// TIA Portal V20 export
FUNCTION "02 T1-A ARUNC HMI" : Void   // FC1202, LAD
TITLE = HMI
{ S7_Optimized_Access := 'TRUE' }
// stored: AutoNumber false, SetENOAutomatically false
BEGIN

REGION Network 1: Reset command interface from HMI in case of time-out
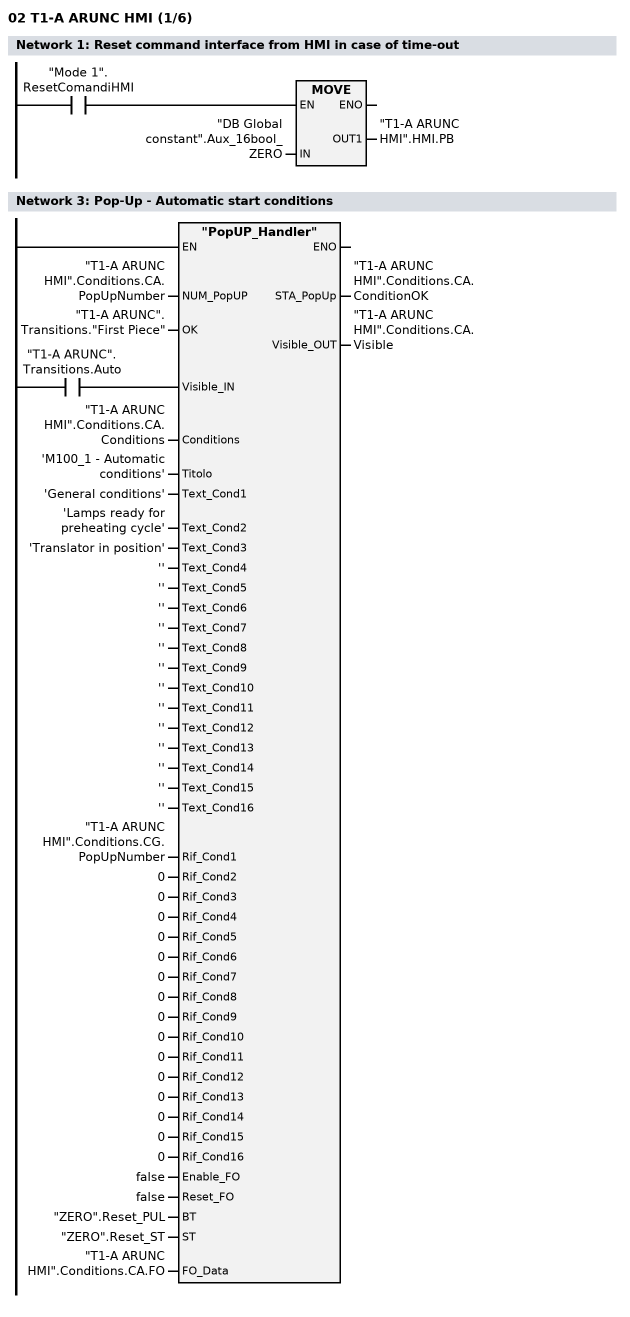
   RUNG wire#powerrail
      Contact( "Mode 1".ResetComandiHMI )
      Move(in := "DB Global constant".Aux_16bool_ZERO, out1 => "T1-A ARUNC HMI".HMI.PB)
   END_RUNG
   // the same network as SCL:
   IF "Mode 1".ResetComandiHMI THEN "T1-A ARUNC HMI".HMI.PB := "DB Global constant".Aux_16bool_ZERO; END_IF;
END_REGION

REGION Network 2: ============ POP UP ============
END_REGION

REGION Network 3: Pop-Up - Automatic start conditions
   RUNG wire#powerrail
      "PopUP_Handler"(Visible_IN := wire#w1, NUM_PopUP := "T1-A ARUNC HMI".Conditions.CA.PopUpNumber, OK := "T1-A ARUNC".Transitions."First Piece", Conditions := "T1-A ARUNC HMI".Conditions.CA.Conditions, Titolo := 'M100_1 - Automatic conditions', Text_Cond1 := 'General conditions', Text_Cond2 := 'Lamps ready for preheating cycle', Text_Cond3 := 'Translator in position', Text_Cond4 := '', Text_Cond5 := '', Text_Cond6 := '', Text_Cond7 := '', Text_Cond8 := '', Text_Cond9 := '', Text_Cond10 := '', Text_Cond11 := '', Text_Cond12 := '', Text_Cond13 := '', Text_Cond14 := '', Text_Cond15 := '', Text_Cond16 := '', Rif_Cond1 := "T1-A ARUNC HMI".Conditions.CG.PopUpNumber, Rif_Cond2 := 0, Rif_Cond3 := 0, Rif_Cond4 := 0, Rif_Cond5 := 0, Rif_Cond6 := 0, Rif_Cond7 := 0, Rif_Cond8 := 0, Rif_Cond9 := 0, Rif_Cond10 := 0, Rif_Cond11 := 0, Rif_Cond12 := 0, Rif_Cond13 := 0, Rif_Cond14 := 0, Rif_Cond15 := 0, Rif_Cond16 := 0, Enable_FO := false, Reset_FO := false, BT := "ZERO".Reset_PUL, ST := "ZERO".Reset_ST, FO_Data := "T1-A ARUNC HMI".Conditions.CA.FO, STA_PopUp => "T1-A ARUNC HMI".Conditions.CA.ConditionOK, Visible_OUT => "T1-A ARUNC HMI".Conditions.CA.Visible)
   END_RUNG
   RUNG wire#powerrail
      Contact( "T1-A ARUNC".Transitions.Auto )
   END_RUNG wire#w1
   // the same network as SCL:
   "PopUP_Handler"(NUM_PopUP := "T1-A ARUNC HMI".Conditions.CA.PopUpNumber,
                   OK := "T1-A ARUNC".Transitions."First Piece",
                   Visible_IN := "T1-A ARUNC".Transitions.Auto,
                   Conditions := "T1-A ARUNC HMI".Conditions.CA.Conditions,
                   Titolo := 'M100_1 - Automatic conditions',
                   Text_Cond1 := 'General conditions',
                   Text_Cond2 := 'Lamps ready for preheating cycle',
                   Text_Cond3 := 'Translator in position',
                   Text_Cond4 := '',
                   Text_Cond5 := '',
                   Text_Cond6 := '',
                   Text_Cond7 := '',
                   Text_Cond8 := '',
                   Text_Cond9 := '',
                   Text_Cond10 := '',
                   Text_Cond11 := '',
                   Text_Cond12 := '',
                   Text_Cond13 := '',
                   Text_Cond14 := '',
                   Text_Cond15 := '',
                   Text_Cond16 := '',
                   Rif_Cond1 := "T1-A ARUNC HMI".Conditions.CG.PopUpNumber,
                   Rif_Cond2 := 0,
                   Rif_Cond3 := 0,
                   Rif_Cond4 := 0,
                   Rif_Cond5 := 0,
                   Rif_Cond6 := 0,
                   Rif_Cond7 := 0,
                   Rif_Cond8 := 0,
                   Rif_Cond9 := 0,
                   Rif_Cond10 := 0,
                   Rif_Cond11 := 0,
                   Rif_Cond12 := 0,
                   Rif_Cond13 := 0,
                   Rif_Cond14 := 0,
                   Rif_Cond15 := 0,
                   Rif_Cond16 := 0,
                   Enable_FO := false,
                   Reset_FO := false,
                   BT := "ZERO".Reset_PUL,
                   ST := "ZERO".Reset_ST,
                   FO_Data := "T1-A ARUNC HMI".Conditions.CA.FO,
                   STA_PopUp => "T1-A ARUNC HMI".Conditions.CA.ConditionOK,
                   Visible_OUT => "T1-A ARUNC HMI".Conditions.CA.Visible);
END_REGION

REGION Network 4: Pop- Up - General conditions
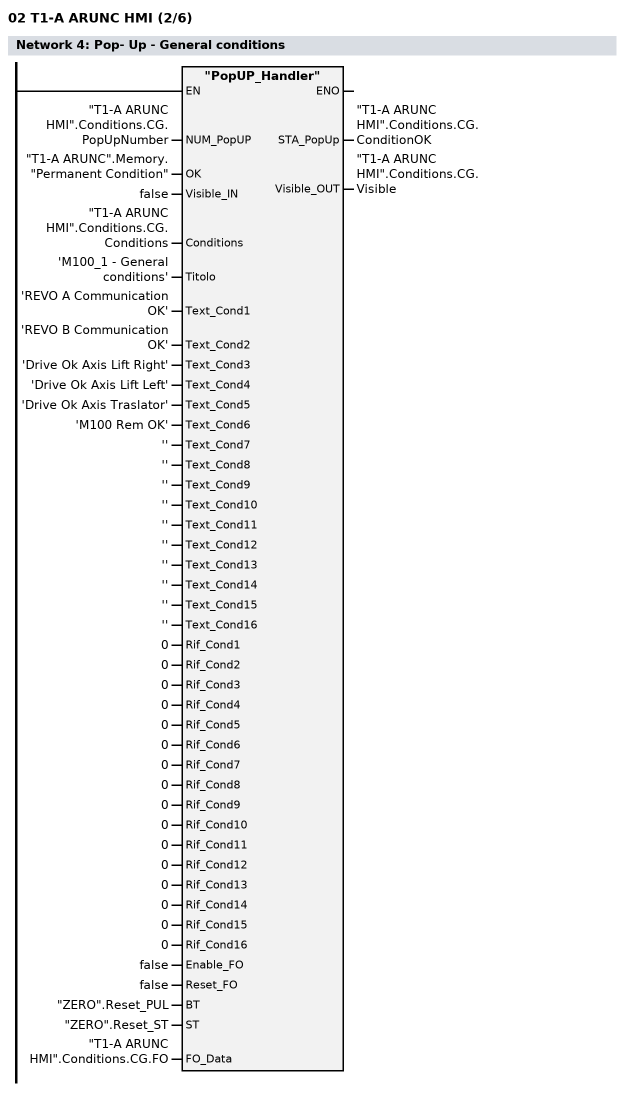
   RUNG wire#powerrail
      "PopUP_Handler"(NUM_PopUP := "T1-A ARUNC HMI".Conditions.CG.PopUpNumber, OK := "T1-A ARUNC".Memory."Permanent Condition", Visible_IN := false, Conditions := "T1-A ARUNC HMI".Conditions.CG.Conditions, Titolo := 'M100_1 - General conditions', Text_Cond1 := 'REVO A Communication OK', Text_Cond2 := 'REVO B Communication OK', Text_Cond3 := 'Drive Ok Axis Lift Right', Text_Cond4 := 'Drive Ok Axis Lift Left', Text_Cond5 := 'Drive Ok Axis Traslator', Text_Cond6 := 'M100 Rem OK', Text_Cond7 := '', Text_Cond8 := '', Text_Cond9 := '', Text_Cond10 := '', Text_Cond11 := '', Text_Cond12 := '', Text_Cond13 := '', Text_Cond14 := '', Text_Cond15 := '', Text_Cond16 := '', Rif_Cond1 := 0, Rif_Cond2 := 0, Rif_Cond3 := 0, Rif_Cond4 := 0, Rif_Cond5 := 0, Rif_Cond6 := 0, Rif_Cond7 := 0, Rif_Cond8 := 0, Rif_Cond9 := 0, Rif_Cond10 := 0, Rif_Cond11 := 0, Rif_Cond12 := 0, Rif_Cond13 := 0, Rif_Cond14 := 0, Rif_Cond15 := 0, Rif_Cond16 := 0, Enable_FO := false, Reset_FO := false, BT := "ZERO".Reset_PUL, ST := "ZERO".Reset_ST, FO_Data := "T1-A ARUNC HMI".Conditions.CG.FO, STA_PopUp => "T1-A ARUNC HMI".Conditions.CG.ConditionOK, Visible_OUT => "T1-A ARUNC HMI".Conditions.CG.Visible)
   END_RUNG
   // the same network as SCL:
   "PopUP_Handler"(NUM_PopUP := "T1-A ARUNC HMI".Conditions.CG.PopUpNumber,
                   OK := "T1-A ARUNC".Memory."Permanent Condition",
                   Visible_IN := false,
                   Conditions := "T1-A ARUNC HMI".Conditions.CG.Conditions,
                   Titolo := 'M100_1 - General conditions',
                   Text_Cond1 := 'REVO A Communication OK',
                   Text_Cond2 := 'REVO B Communication OK',
                   Text_Cond3 := 'Drive Ok Axis Lift Right',
                   Text_Cond4 := 'Drive Ok Axis Lift Left',
                   Text_Cond5 := 'Drive Ok Axis Traslator',
                   Text_Cond6 := 'M100 Rem OK',
                   Text_Cond7 := '',
                   Text_Cond8 := '',
                   Text_Cond9 := '',
                   Text_Cond10 := '',
                   Text_Cond11 := '',
                   Text_Cond12 := '',
                   Text_Cond13 := '',
                   Text_Cond14 := '',
                   Text_Cond15 := '',
                   Text_Cond16 := '',
                   Rif_Cond1 := 0,
                   Rif_Cond2 := 0,
                   Rif_Cond3 := 0,
                   Rif_Cond4 := 0,
                   Rif_Cond5 := 0,
                   Rif_Cond6 := 0,
                   Rif_Cond7 := 0,
                   Rif_Cond8 := 0,
                   Rif_Cond9 := 0,
                   Rif_Cond10 := 0,
                   Rif_Cond11 := 0,
                   Rif_Cond12 := 0,
                   Rif_Cond13 := 0,
                   Rif_Cond14 := 0,
                   Rif_Cond15 := 0,
                   Rif_Cond16 := 0,
                   Enable_FO := false,
                   Reset_FO := false,
                   BT := "ZERO".Reset_PUL,
                   ST := "ZERO".Reset_ST,
                   FO_Data := "T1-A ARUNC HMI".Conditions.CG.FO,
                   STA_PopUp => "T1-A ARUNC HMI".Conditions.CG.ConditionOK,
                   Visible_OUT => "T1-A ARUNC HMI".Conditions.CG.Visible);
END_REGION

REGION Network 5: PopUP - Cycle start conditions
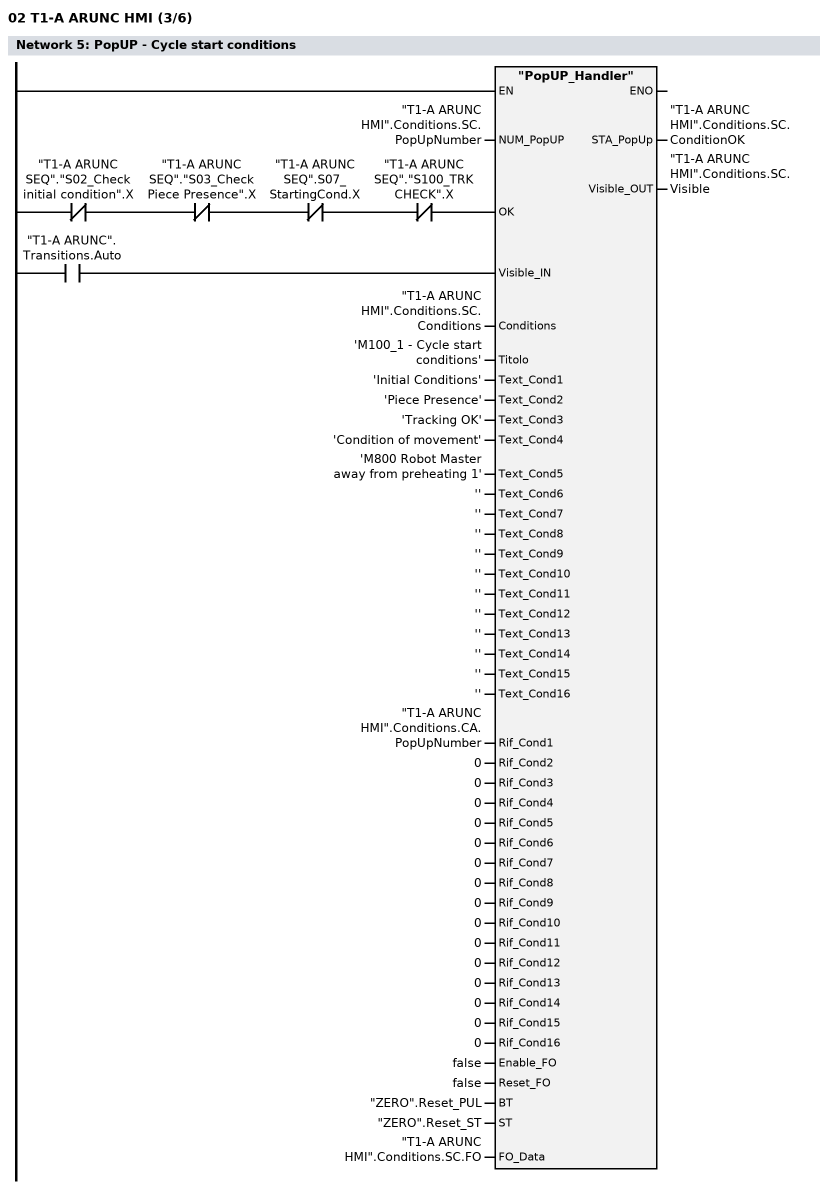
   RUNG wire#powerrail
      "PopUP_Handler"(OK := wire#w1, Visible_IN := wire#w2, NUM_PopUP := "T1-A ARUNC HMI".Conditions.SC.PopUpNumber, Conditions := "T1-A ARUNC HMI".Conditions.SC.Conditions, Titolo := 'M100_1 - Cycle start conditions', Text_Cond1 := 'Initial Conditions', Text_Cond2 := 'Piece Presence', Text_Cond3 := 'Tracking OK', Text_Cond4 := 'Condition of movement', Text_Cond5 := 'M800 Robot Master away from preheating 1', Text_Cond6 := '', Text_Cond7 := '', Text_Cond8 := '', Text_Cond9 := '', Text_Cond10 := '', Text_Cond11 := '', Text_Cond12 := '', Text_Cond13 := '', Text_Cond14 := '', Text_Cond15 := '', Text_Cond16 := '', Rif_Cond1 := "T1-A ARUNC HMI".Conditions.CA.PopUpNumber, Rif_Cond2 := 0, Rif_Cond3 := 0, Rif_Cond4 := 0, Rif_Cond5 := 0, Rif_Cond6 := 0, Rif_Cond7 := 0, Rif_Cond8 := 0, Rif_Cond9 := 0, Rif_Cond10 := 0, Rif_Cond11 := 0, Rif_Cond12 := 0, Rif_Cond13 := 0, Rif_Cond14 := 0, Rif_Cond15 := 0, Rif_Cond16 := 0, Enable_FO := false, Reset_FO := false, BT := "ZERO".Reset_PUL, ST := "ZERO".Reset_ST, FO_Data := "T1-A ARUNC HMI".Conditions.SC.FO, STA_PopUp => "T1-A ARUNC HMI".Conditions.SC.ConditionOK, Visible_OUT => "T1-A ARUNC HMI".Conditions.SC.Visible)
   END_RUNG
   RUNG wire#powerrail
      I_Contact( "T1-A ARUNC SEQ"."S02_Check initial condition".X )
      I_Contact( "T1-A ARUNC SEQ"."S03_Check Piece Presence".X )
      I_Contact( "T1-A ARUNC SEQ".S07_StartingCond.X )
      I_Contact( "T1-A ARUNC SEQ"."S100_TRK CHECK".X )
   END_RUNG wire#w1
   RUNG wire#powerrail
      Contact( "T1-A ARUNC".Transitions.Auto )
   END_RUNG wire#w2
   // the same network as SCL:
   "PopUP_Handler"(NUM_PopUP := "T1-A ARUNC HMI".Conditions.SC.PopUpNumber,
                   OK := NOT "T1-A ARUNC SEQ"."S02_Check initial condition".X AND NOT "T1-A ARUNC SEQ"."S03_Check Piece Presence".X AND NOT "T1-A ARUNC SEQ".S07_StartingCond.X AND NOT "T1-A ARUNC SEQ"."S100_TRK CHECK".X,
                   Visible_IN := "T1-A ARUNC".Transitions.Auto,
                   Conditions := "T1-A ARUNC HMI".Conditions.SC.Conditions,
                   Titolo := 'M100_1 - Cycle start conditions',
                   Text_Cond1 := 'Initial Conditions',
                   Text_Cond2 := 'Piece Presence',
                   Text_Cond3 := 'Tracking OK',
                   Text_Cond4 := 'Condition of movement',
                   Text_Cond5 := 'M800 Robot Master away from preheating 1',
                   Text_Cond6 := '',
                   Text_Cond7 := '',
                   Text_Cond8 := '',
                   Text_Cond9 := '',
                   Text_Cond10 := '',
                   Text_Cond11 := '',
                   Text_Cond12 := '',
                   Text_Cond13 := '',
                   Text_Cond14 := '',
                   Text_Cond15 := '',
                   Text_Cond16 := '',
                   Rif_Cond1 := "T1-A ARUNC HMI".Conditions.CA.PopUpNumber,
                   Rif_Cond2 := 0,
                   Rif_Cond3 := 0,
                   Rif_Cond4 := 0,
                   Rif_Cond5 := 0,
                   Rif_Cond6 := 0,
                   Rif_Cond7 := 0,
                   Rif_Cond8 := 0,
                   Rif_Cond9 := 0,
                   Rif_Cond10 := 0,
                   Rif_Cond11 := 0,
                   Rif_Cond12 := 0,
                   Rif_Cond13 := 0,
                   Rif_Cond14 := 0,
                   Rif_Cond15 := 0,
                   Rif_Cond16 := 0,
                   Enable_FO := false,
                   Reset_FO := false,
                   BT := "ZERO".Reset_PUL,
                   ST := "ZERO".Reset_ST,
                   FO_Data := "T1-A ARUNC HMI".Conditions.SC.FO,
                   STA_PopUp => "T1-A ARUNC HMI".Conditions.SC.ConditionOK,
                   Visible_OUT => "T1-A ARUNC HMI".Conditions.SC.Visible);
END_REGION

REGION Network 6: Pop-Up - Conditions of movement UP
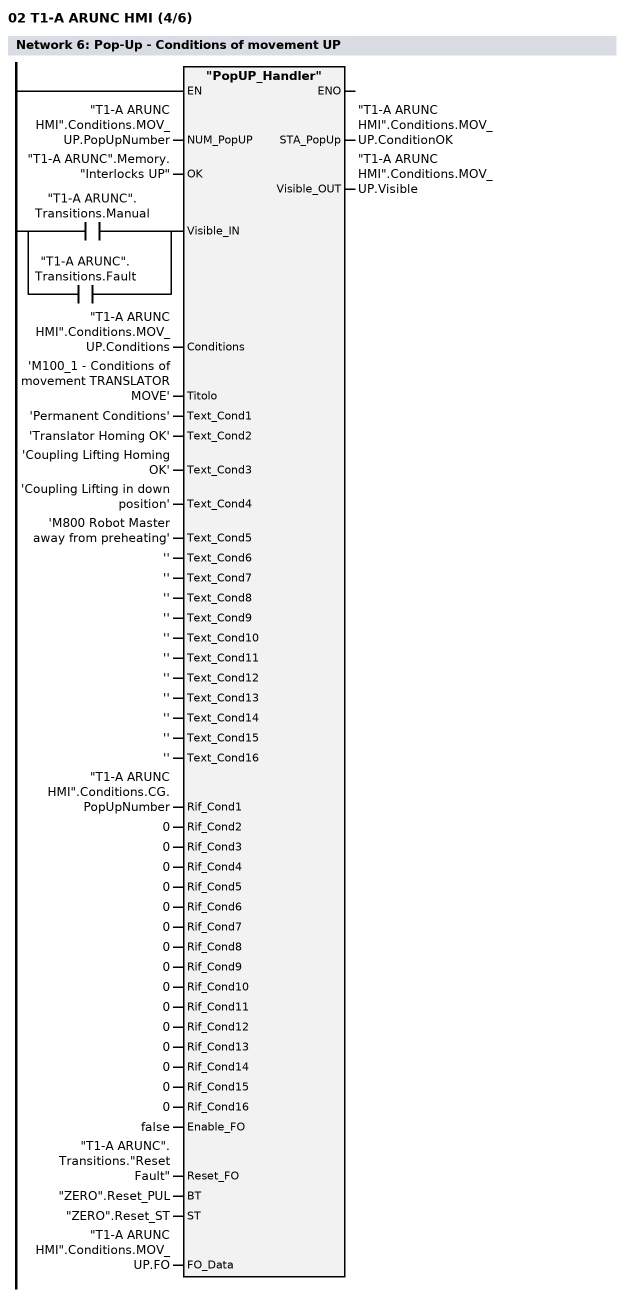
   RUNG wire#powerrail
      "PopUP_Handler"(Visible_IN := wire#w1, NUM_PopUP := "T1-A ARUNC HMI".Conditions.MOV_UP.PopUpNumber, OK := "T1-A ARUNC".Memory."Interlocks UP", Conditions := "T1-A ARUNC HMI".Conditions.MOV_UP.Conditions, Titolo := 'M100_1 - Conditions of movement TRANSLATOR MOVE', Text_Cond1 := 'Permanent Conditions', Text_Cond2 := 'Translator Homing OK', Text_Cond3 := 'Coupling Lifting Homing OK', Text_Cond4 := 'Coupling Lifting in down position', Text_Cond5 := 'M800 Robot Master away from preheating', Text_Cond6 := '', Text_Cond7 := '', Text_Cond8 := '', Text_Cond9 := '', Text_Cond10 := '', Text_Cond11 := '', Text_Cond12 := '', Text_Cond13 := '', Text_Cond14 := '', Text_Cond15 := '', Text_Cond16 := '', Rif_Cond1 := "T1-A ARUNC HMI".Conditions.CG.PopUpNumber, Rif_Cond2 := 0, Rif_Cond3 := 0, Rif_Cond4 := 0, Rif_Cond5 := 0, Rif_Cond6 := 0, Rif_Cond7 := 0, Rif_Cond8 := 0, Rif_Cond9 := 0, Rif_Cond10 := 0, Rif_Cond11 := 0, Rif_Cond12 := 0, Rif_Cond13 := 0, Rif_Cond14 := 0, Rif_Cond15 := 0, Rif_Cond16 := 0, Enable_FO := false, Reset_FO := "T1-A ARUNC".Transitions."Reset Fault", BT := "ZERO".Reset_PUL, ST := "ZERO".Reset_ST, FO_Data := "T1-A ARUNC HMI".Conditions.MOV_UP.FO, STA_PopUp => "T1-A ARUNC HMI".Conditions.MOV_UP.ConditionOK, Visible_OUT => "T1-A ARUNC HMI".Conditions.MOV_UP.Visible)
   END_RUNG
   RUNG wire#powerrail
      Contact( "T1-A ARUNC".Transitions.Manual )
   END_RUNG wire#w1
   RUNG wire#powerrail
      Contact( "T1-A ARUNC".Transitions.Fault )
   END_RUNG wire#w1
   // the same network as SCL:
   "PopUP_Handler"(NUM_PopUP := "T1-A ARUNC HMI".Conditions.MOV_UP.PopUpNumber,
                   OK := "T1-A ARUNC".Memory."Interlocks UP",
                   Visible_IN := "T1-A ARUNC".Transitions.Manual OR "T1-A ARUNC".Transitions.Fault,
                   Conditions := "T1-A ARUNC HMI".Conditions.MOV_UP.Conditions,
                   Titolo := 'M100_1 - Conditions of movement TRANSLATOR MOVE',
                   Text_Cond1 := 'Permanent Conditions',
                   Text_Cond2 := 'Translator Homing OK',
                   Text_Cond3 := 'Coupling Lifting Homing OK',
                   Text_Cond4 := 'Coupling Lifting in down position',
                   Text_Cond5 := 'M800 Robot Master away from preheating',
                   Text_Cond6 := '',
                   Text_Cond7 := '',
                   Text_Cond8 := '',
                   Text_Cond9 := '',
                   Text_Cond10 := '',
                   Text_Cond11 := '',
                   Text_Cond12 := '',
                   Text_Cond13 := '',
                   Text_Cond14 := '',
                   Text_Cond15 := '',
                   Text_Cond16 := '',
                   Rif_Cond1 := "T1-A ARUNC HMI".Conditions.CG.PopUpNumber,
                   Rif_Cond2 := 0,
                   Rif_Cond3 := 0,
                   Rif_Cond4 := 0,
                   Rif_Cond5 := 0,
                   Rif_Cond6 := 0,
                   Rif_Cond7 := 0,
                   Rif_Cond8 := 0,
                   Rif_Cond9 := 0,
                   Rif_Cond10 := 0,
                   Rif_Cond11 := 0,
                   Rif_Cond12 := 0,
                   Rif_Cond13 := 0,
                   Rif_Cond14 := 0,
                   Rif_Cond15 := 0,
                   Rif_Cond16 := 0,
                   Enable_FO := false,
                   Reset_FO := "T1-A ARUNC".Transitions."Reset Fault",
                   BT := "ZERO".Reset_PUL,
                   ST := "ZERO".Reset_ST,
                   FO_Data := "T1-A ARUNC HMI".Conditions.MOV_UP.FO,
                   STA_PopUp => "T1-A ARUNC HMI".Conditions.MOV_UP.ConditionOK,
                   Visible_OUT => "T1-A ARUNC HMI".Conditions.MOV_UP.Visible);
END_REGION

REGION Network 7: ============ HMI STATE ============
END_REGION

REGION Network 8: HMI Status - Aruncator
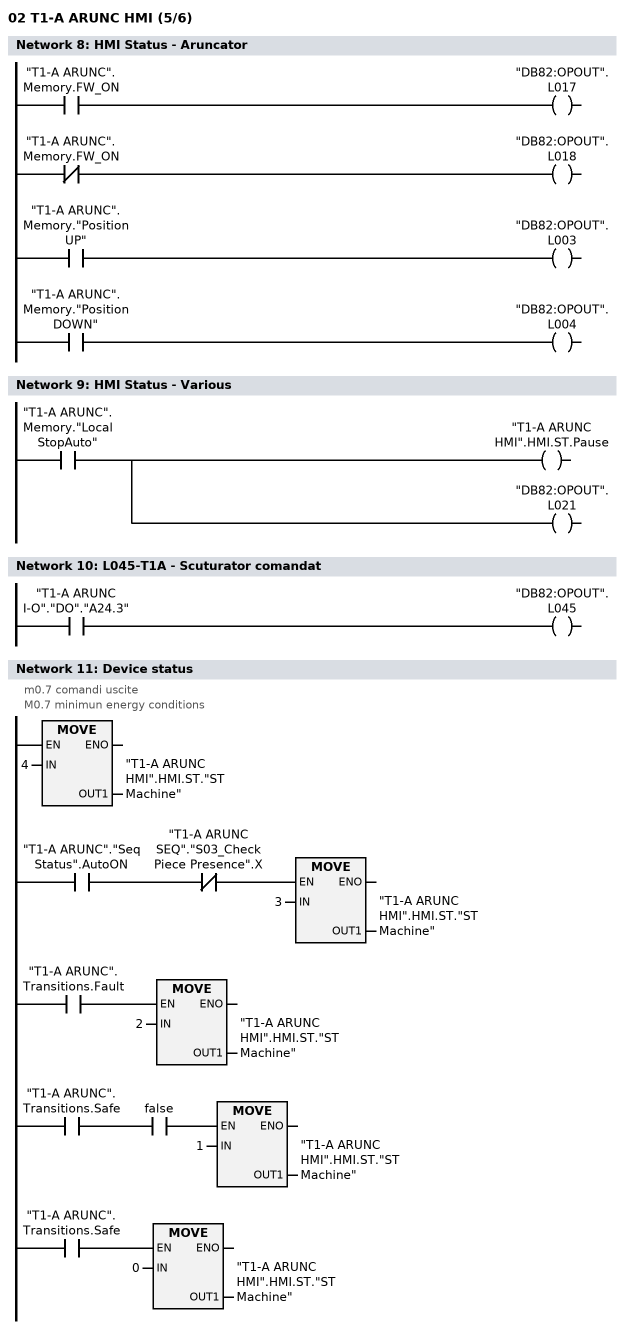
   RUNG wire#powerrail
      Contact( "T1-A ARUNC".Memory.FW_ON )
      Coil( "DB82:OPOUT".L017 )
   END_RUNG
   RUNG wire#powerrail
      I_Contact( "T1-A ARUNC".Memory.FW_ON )
      Coil( "DB82:OPOUT".L018 )
   END_RUNG
   RUNG wire#powerrail
      Contact( "T1-A ARUNC".Memory."Position UP" )
      Coil( "DB82:OPOUT".L003 )
   END_RUNG
   RUNG wire#powerrail
      Contact( "T1-A ARUNC".Memory."Position DOWN" )
      Coil( "DB82:OPOUT".L004 )
   END_RUNG
   // the same network as SCL:
   "DB82:OPOUT".L017 := "T1-A ARUNC".Memory.FW_ON;
   "DB82:OPOUT".L018 := NOT "T1-A ARUNC".Memory.FW_ON;
   "DB82:OPOUT".L003 := "T1-A ARUNC".Memory."Position UP";
   "DB82:OPOUT".L004 := "T1-A ARUNC".Memory."Position DOWN";
END_REGION

REGION Network 9: HMI Status - Various
   RUNG wire#powerrail
      Contact( "T1-A ARUNC".Memory."Local StopAuto" )
      wire#w1
      Coil( "T1-A ARUNC HMI".HMI.ST.Pause )
   END_RUNG
   RUNG wire#w1
      Coil( "DB82:OPOUT".L021 )
   END_RUNG
   // the same network as SCL:
   "T1-A ARUNC HMI".HMI.ST.Pause := "T1-A ARUNC".Memory."Local StopAuto";
   "DB82:OPOUT".L021 := "T1-A ARUNC".Memory."Local StopAuto";
END_REGION

REGION Network 10: L045-T1A - Scuturator comandat
   RUNG wire#powerrail
      Contact( "T1-A ARUNC I-O"."DO"."A24.3" )
      Coil( "DB82:OPOUT".L045 )
   END_RUNG
   // the same network as SCL:
   "DB82:OPOUT".L045 := "T1-A ARUNC I-O"."DO"."A24.3";
END_REGION

REGION Network 11: Device status
   // m0.7 comandi uscite
   // M0.7 minimun energy conditions
   RUNG wire#powerrail
      Move(in := 4, out1 => "T1-A ARUNC HMI".HMI.ST."ST Machine")
   END_RUNG
   RUNG wire#powerrail
      Contact( "T1-A ARUNC"."Seq Status".AutoON )
      I_Contact( "T1-A ARUNC SEQ"."S03_Check Piece Presence".X )
      Move(in := 3, out1 => "T1-A ARUNC HMI".HMI.ST."ST Machine")
   END_RUNG
   RUNG wire#powerrail
      Contact( "T1-A ARUNC".Transitions.Fault )
      Move(in := 2, out1 => "T1-A ARUNC HMI".HMI.ST."ST Machine")
   END_RUNG
   RUNG wire#powerrail
      Contact( "T1-A ARUNC".Transitions.Safe )
      Contact( false )
      Move(in := 1, out1 => "T1-A ARUNC HMI".HMI.ST."ST Machine")
   END_RUNG
   RUNG wire#powerrail
      Contact( "T1-A ARUNC".Transitions.Safe )
      Move(in := 0, out1 => "T1-A ARUNC HMI".HMI.ST."ST Machine")
   END_RUNG
   // the same network as SCL:
   "T1-A ARUNC HMI".HMI.ST."ST Machine" := 4;
   IF "T1-A ARUNC"."Seq Status".AutoON AND NOT "T1-A ARUNC SEQ"."S03_Check Piece Presence".X THEN
       "T1-A ARUNC HMI".HMI.ST."ST Machine" := 3;
   END_IF;
   IF "T1-A ARUNC".Transitions.Fault THEN "T1-A ARUNC HMI".HMI.ST."ST Machine" := 2; END_IF;
   IF "T1-A ARUNC".Transitions.Safe AND false THEN "T1-A ARUNC HMI".HMI.ST."ST Machine" := 1; END_IF;
   IF "T1-A ARUNC".Transitions.Safe THEN "T1-A ARUNC HMI".HMI.ST."ST Machine" := 0; END_IF;
END_REGION

REGION Network 12: Sequencer status
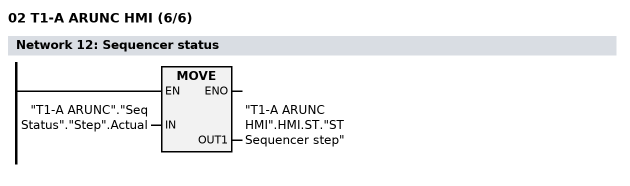
   RUNG wire#powerrail
      Move(in := "T1-A ARUNC"."Seq Status"."Step".Actual, out1 => "T1-A ARUNC HMI".HMI.ST."ST Sequencer step")
   END_RUNG
   // the same network as SCL:
   "T1-A ARUNC HMI".HMI.ST."ST Sequencer step" := "T1-A ARUNC"."Seq Status"."Step".Actual;
END_REGION
END_FUNCTION
